// Struckig
// Copyright (C) 2022 Stefan Besler

// This program is free software: you can redistribute it and/or modify
// it under the terms of the GNU General Public License as published by
// the Free Software Foundation, either version 3 of the License, or
// (at your option) any later version.

// This program is distributed in the hope that it will be useful,
// but WITHOUT ANY WARRANTY; without even the implied warranty of
// MERCHANTABILITY or FITNESS FOR A PARTICULAR PURPOSE.  See the
// GNU General Public License for more details.
//
// You should have received a copy of the GNU General Public License
// along with THIS PROGRAM.  IF NOT, see <http://www.gnu.org/licenses/>.
{attribute 'conditionalshow_all_locals'}
/// Convenience wrapper for single-DoF trajectory generation.
/// This function block forwards all calls to an internal `Otg` instance with `Dofs = 1`.
/// Use this block when your application controls exactly one axis and you want
/// scalar I/O instead of vectors.
///
/// ```st
/// otg1(
///   CycleTime := 0.001,
///   ControlInterface := ControlInterfaceType.Position,
///   Synchronization := SynchronizationType.TimeSync
/// );
/// Axis.Setpoint := otg1.NewPosition;
/// ```
FUNCTION_BLOCK Otg1 IMPLEMENTS IOtg
VAR_INPUT
  CycleTime : LREAL;
  ControlInterface : ControlInterfaceType := ControlInterfaceType.Position; //< The default position interface controls the full kinematic state.
  Synchronization : SynchronizationType := SynchronizationType.TimeSync; //< Synchronization behavior of multiple DoFs
  PerDofControlInterface : ControlInterfaceType; //< Per-DoF control interface (overwrites global ControlInterface)
  PerDofSynchronization :  SynchronizationType; //< Per-DoF synchronization (overwrites global Synchronization)
  Discretization : DiscretizationType; //< Whether the duration should be a discrete multiple of the control cycle (off by default)
  CurrentPosition, CurrentVelocity, CurrentAcceleration : LREAL; //< Current state
  TargetPosition, TargetVelocity, TargetAcceleration : LREAL; //< Target state
  MaxVelocity, MaxAcceleration, MaxJerk : LREAL; //< Kinematic constraints
  MinVelocity, MinAcceleration : LREAL; //< Optional kindematic constraints
  MinDuration : LREAL := 0; //< Optional minimum duration of a trajectory. This is only considered if the Synchronization type is not none
  EnableAutoPropagate : BOOL; //< If set to true, PassOutputToInput is automatically called internally after calling the function block's body
  SmoothBrake : BOOL := ParameterList.SmoothBrake; //< See Otg.SmoothBrake
END_VAR
VAR_OUTPUT
  NewPosition, NewVelocity, NewAcceleration, NewJerk : LREAL;
  NewCalculation : BOOL; //< Was a new trajectory calculation performed in the last cycle?
  CurrentTime : LREAL; //< Time elapsed on the current trajectory in seconds.
END_VAR
VAR
  _otg : Otg(0,0);
END_VAR

_otg.PerDofControlInterface[0] := PerDofControlInterface;
_otg.PerDofSynchronization[0] := PerDofSynchronization;
_otg.Discretization := Discretization;
_otg.CurrentPosition[0] := CurrentPosition;
_otg.CurrentVelocity[0] := CurrentVelocity;
_otg.CurrentAcceleration[0] := CurrentAcceleration;
_otg.TargetPosition[0] := TargetPosition;
_otg.TargetVelocity[0] := TargetVelocity;
_otg.TargetAcceleration[0] := TargetAcceleration;
_otg.MaxVelocity[0] := MaxVelocity;
_otg.MaxAcceleration[0] := MaxAcceleration;
_otg.MaxJerk[0] := MaxJerk;
_otg.MinVelocity[0] := MinVelocity;
_otg.MinAcceleration[0] := MinAcceleration;
_otg.MinDuration := MinDuration;
_otg.EnableAutoPropagate := EnableAutoPropagate;
_otg.SmoothBrake := SmoothBrake;

_otg(CycleTime := CycleTime,
     Dofs := 1,
     ControlInterface := ControlInterface,
     Synchronization := Synchronization);
     
CurrentPosition := _otg.CurrentPosition[0];
CurrentVelocity := _otg.CurrentVelocity[0];
CurrentAcceleration := _otg.CurrentAcceleration[0];     
NewPosition := _otg.NewPosition[0];
NewVelocity := _otg.NewVelocity[0];
NewAcceleration := _otg.NewAcceleration[0];
NewJerk := _otg.NewJerk[0];
CurrentTime := _otg.CurrentTime;

/// \copydoc Struckig.Otg#AtTime
{attribute 'conditionalshow'}
METHOD AtTime
VAR_INPUT
  t : LREAL;
  new_position : POINTER TO LREAL;
  new_velocity : POINTER TO LREAL;
  new_acceleration : POINTER TO LREAL;
  new_jerk : POINTER TO LREAL;
  new_section : POINTER TO INT;
END_VAR
_otg.AtTime(t, new_position, new_velocity, new_acceleration, new_jerk, new_section);
END_METHOD

/// \copydoc Struckig.Otg#AtTime1
{attribute 'conditionalshow'}
METHOD AtTime1
VAR_INPUT
  t : LREAL;
  new_position : REFERENCE TO LREAL;
  new_velocity : REFERENCE TO LREAL;
  new_acceleration : REFERENCE TO LREAL;
  new_jerk : REFERENCE TO LREAL;  
END_VAR
_otg.AtTime1(t, new_position, new_velocity, new_acceleration, new_jerk);
END_METHOD

/// \copydoc Struckig.Otg#Cyclic
METHOD Cyclic
VAR_INPUT
END_VAR
_otg();
END_METHOD

/// \copydoc Struckig.Otg#Duration
PROPERTY Duration : LREAL
GET
Duration := _otg.Duration;
END_GET
END_PROPERTY

/// \copydoc Struckig.Otg#ErrorCode
METHOD ErrorCode : TrajectoryErrorCode
VAR_INPUT
END_VAR
ErrorCode := _otg.ErrorCode();
END_METHOD

/// \copydoc Struckig.Otg#ErrorMessage
METHOD ErrorMessage : STRING(255)
VAR_INPUT
END_VAR
ErrorMessage := _otg.ErrorMessage();
END_METHOD

METHOD FB_init : BOOL
VAR_INPUT
	bInitRetains : BOOL; // if TRUE, the retain variables are initialized (warm start / cold start)
	bInCopyCode : BOOL;  // if TRUE, the instance afterwards gets moved into the copy code (online change)
  cycletime : LREAL;
END_VAR
_otg.FB_init(bInitRetains, bInCopyCode, cycletime, 1);
THIS^.CycleTime := cycletime;
END_METHOD

/// \copydoc Struckig.Otg#PassOutputToInput
METHOD PassOutputToInput
VAR_INPUT
END_VAR
_otg.PassOutputToInput();
END_METHOD

/// \copydoc Struckig.Otg#Reset
METHOD Reset
VAR_INPUT
END_VAR
_otg.Reset();
END_METHOD

/// \copydoc Struckig.Otg#State
PROPERTY State : TrajectoryState
GET
State := _otg.State;
END_GET
END_PROPERTY

/// \copydoc Struckig.Otg#ValidateInput
{attribute 'conditionalshow'}
METHOD ValidateInput : BOOL
VAR_INPUT
  checkCurrentStateWithinLimits : BOOL;
  checkTargetStateWithinLimits : BOOL;
END_VAR
_otg.ValidateInput(checkCurrentStateWithinLimits, checkTargetStateWithinLimits);
END_METHOD

END_FUNCTION_BLOCK

(* stored: Version 1.1.0.1
   POU Otg1: Id {9885581d-fa47-4155-a97e-9f730ee0a51b}, SpecialFunc None
   Method AtTime: Id {a520beb5-151c-42d0-b2df-d1a48984d915}
   Method AtTime1: Id {1d694463-453a-4697-a59a-2e7b7e0e0ffd}
   Method Cyclic: Id {222cfd84-0828-4551-b3bf-cdb6fa696da0}
   Property Duration: Id {c500a90d-2d0a-4395-8368-a7e5a4ac6445}
   Get Get: Id {4d73abcd-1d4b-4970-898c-c561217a1ac1}
   Method ErrorCode: Id {d66ae977-1948-45e1-af4d-d17d8482ba05}
   Method ErrorMessage: Id {cf0cfe69-ca56-489c-9f3b-08d7e760c4e8}
   Method FB_init: Id {b7cb1bcc-2fba-472d-8488-be869d5cd5c0}
   Method PassOutputToInput: Id {d24bcd13-2f63-4f99-8654-eee02ba9397a}
   Method Reset: Id {f6006d6a-8fe6-4e6f-b876-0bd4c55c24d1}
   Property State: Id {b5ac2802-49ba-47cc-be5c-251e2733bfd0}
   Get Get: Id {1e97f762-4d10-4dd6-8a07-2ee620b245a0}
   Method ValidateInput: Id {6d9acfaa-b45e-458e-bbca-53ad7d22ebed} *)
